% RSLogix 500 project PROJECT 4.RSS, saved by version 8.30.00.16 %
PROJECT "500"    % processor: Bul.1763 MicroLogix 1100 Series B %

PROGRAM FILES
  LAD 2 "MAIN"  4 rungs
  LAD 3 "IO"  7 rungs  % Digital Input %
  LAD 4 "CTRL"  13 rungs
  LAD 8 "CYCLE"  6 rungs

DATA FILES
  O0 OUTPUT  4 elements
  I1 INPUT  6 elements
  S2 STATUS  66 elements
  B3 BINARY  2 elements
  T4 TIMER  3 elements
  C5 COUNTER  1 elements
  R6 CONTROL  1 elements
  N7 INTEGER  1 elements
  F8 FLOAT  1 elements

LADDER 2 "MAIN"
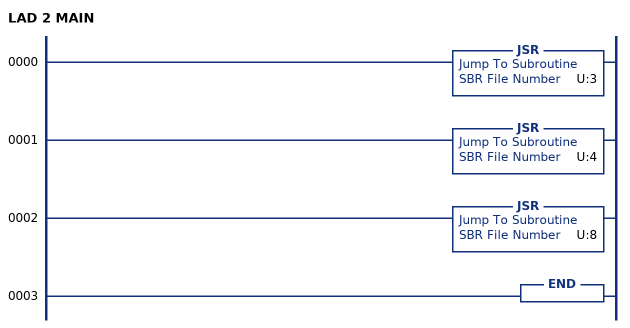
% Rung: 0 %
SOR JSR U:3 EOR
% Rung: 1 %
SOR JSR U:4 EOR
% Rung: 2 %
SOR JSR U:8 EOR
% Rung: 3 %
SOR END EOR

LADDER 3 "IO"    % Digital Input %
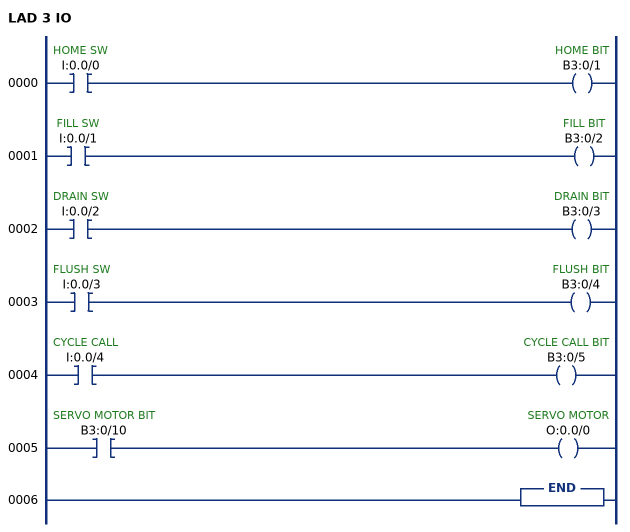
% Rung: 0 %
SOR XIC I:0.0/0 OTE B3:0/1 EOR
%   I:0.0/0  "HOME SW" %
%   B3:0/1  "HOME BIT" %
% Rung: 1 %
SOR XIC I:0.0/1 OTE B3:0/2 EOR
%   I:0.0/1  "FILL SW" %
%   B3:0/2  "FILL BIT" %
% Rung: 2 %
SOR XIC I:0.0/2 OTE B3:0/3 EOR
%   I:0.0/2  "DRAIN SW" %
%   B3:0/3  "DRAIN BIT" %
% Rung: 3 %
SOR XIC I:0.0/3 OTE B3:0/4 EOR
%   I:0.0/3  "FLUSH SW" %
%   B3:0/4  "FLUSH BIT" %
% Rung: 4 %
SOR XIC I:0.0/4 OTE B3:0/5 EOR
%   I:0.0/4  "CYCLE CALL" %
%   B3:0/5  "CYCLE CALL BIT" %
% Rung: 5 %
SOR XIC B3:0/10 OTE O:0.0/0 EOR
%   B3:0/10  "SERVO MOTOR BIT" %
%   O:0.0/0  "SERVO MOTOR" %
% Rung: 6 %
SOR END EOR

LADDER 4 "CTRL"
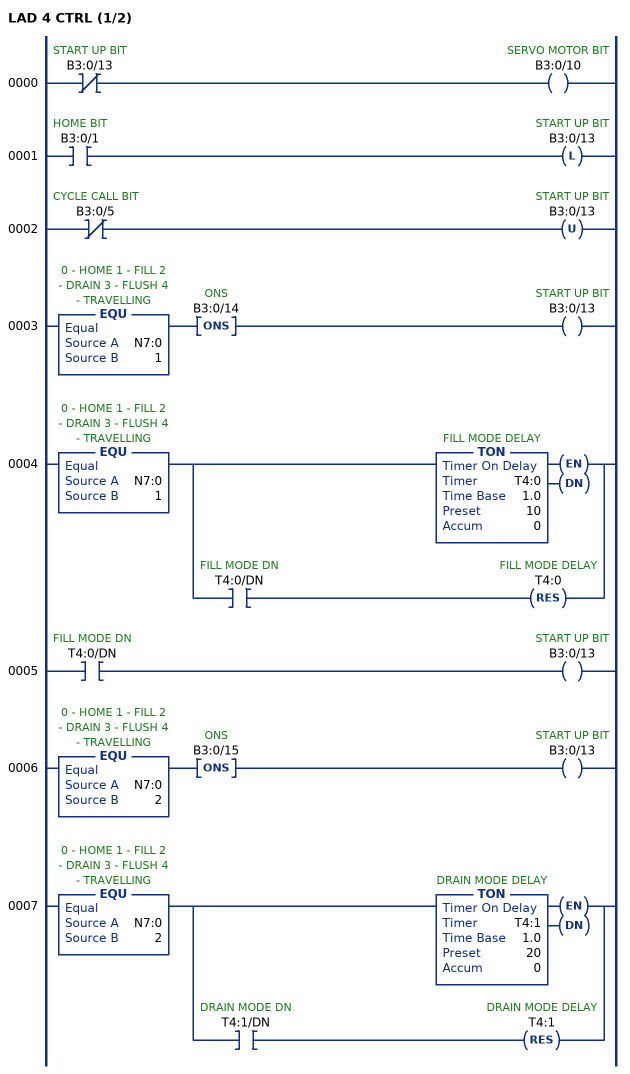
% Rung: 0 %
SOR XIO B3:0/13 OTE B3:0/10 EOR
%   B3:0/13  "START UP BIT" %
%   B3:0/10  "SERVO MOTOR BIT" %
% Rung: 1 %
SOR XIC B3:0/1 OTL B3:0/13 EOR
%   B3:0/1  "HOME BIT" %
%   B3:0/13  "START UP BIT" %
% Rung: 2 %
SOR XIO B3:0/5 OTU B3:0/13 EOR
%   B3:0/5  "CYCLE CALL BIT" %
%   B3:0/13  "START UP BIT" %
% Rung: 3 %
SOR EQU N7:0 1 ONS B3:0/14 OTE B3:0/13 EOR
%   N7:0  "0 - HOME 1 - FILL 2 - DRAIN 3 - FLUSH 4 - TRAVELLING" %
%   B3:0/14  "ONS" %
%   B3:0/13  "START UP BIT" %
% Rung: 4 %
SOR EQU N7:0 1 BST TON T4:0 1.0 10 0 NXB XIC T4:0/DN RES T4:0 BND EOR
%   N7:0  "0 - HOME 1 - FILL 2 - DRAIN 3 - FLUSH 4 - TRAVELLING" %
%   T4:0  "FILL MODE DELAY" %
%   T4:0/DN  "FILL MODE DN" %
% Rung: 5 %
SOR XIC T4:0/DN OTE B3:0/13 EOR
%   T4:0/DN  "FILL MODE DN" %
%   B3:0/13  "START UP BIT" %
% Rung: 6 %
SOR EQU N7:0 2 ONS B3:0/15 OTE B3:0/13 EOR
%   N7:0  "0 - HOME 1 - FILL 2 - DRAIN 3 - FLUSH 4 - TRAVELLING" %
%   B3:0/15  "ONS" %
%   B3:0/13  "START UP BIT" %
% Rung: 7 %
SOR EQU N7:0 2 BST TON T4:1 1.0 20 0 NXB XIC T4:1/DN RES T4:1 BND EOR
%   N7:0  "0 - HOME 1 - FILL 2 - DRAIN 3 - FLUSH 4 - TRAVELLING" %
%   T4:1  "DRAIN MODE DELAY" %
%   T4:1/DN  "DRAIN MODE DN" %

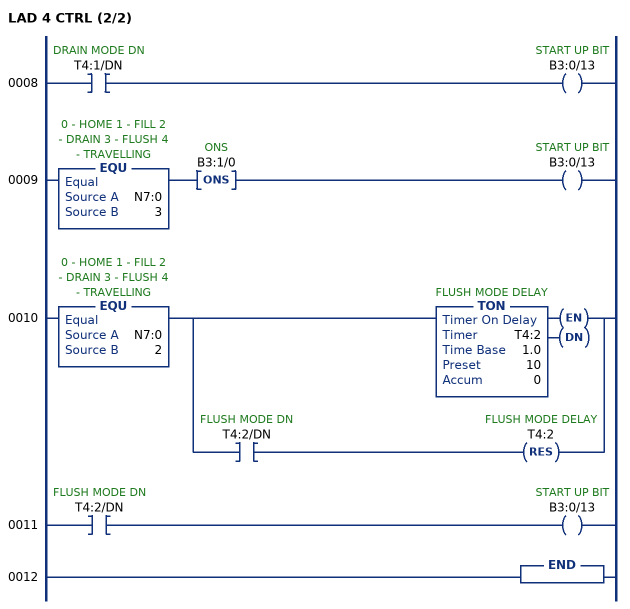
% Rung: 8 %
SOR XIC T4:1/DN OTE B3:0/13 EOR
%   T4:1/DN  "DRAIN MODE DN" %
%   B3:0/13  "START UP BIT" %
% Rung: 9 %
SOR EQU N7:0 3 ONS B3:1/0 OTE B3:0/13 EOR
%   N7:0  "0 - HOME 1 - FILL 2 - DRAIN 3 - FLUSH 4 - TRAVELLING" %
%   B3:1/0  "ONS" %
%   B3:0/13  "START UP BIT" %
% Rung: 10 %
SOR EQU N7:0 2 BST TON T4:2 1.0 10 0 NXB XIC T4:2/DN RES T4:2 BND EOR
%   N7:0  "0 - HOME 1 - FILL 2 - DRAIN 3 - FLUSH 4 - TRAVELLING" %
%   T4:2  "FLUSH MODE DELAY" %
%   T4:2/DN  "FLUSH MODE DN" %
% Rung: 11 %
SOR XIC T4:2/DN OTE B3:0/13 EOR
%   T4:2/DN  "FLUSH MODE DN" %
%   B3:0/13  "START UP BIT" %
% Rung: 12 %
SOR END EOR

LADDER 8 "CYCLE"
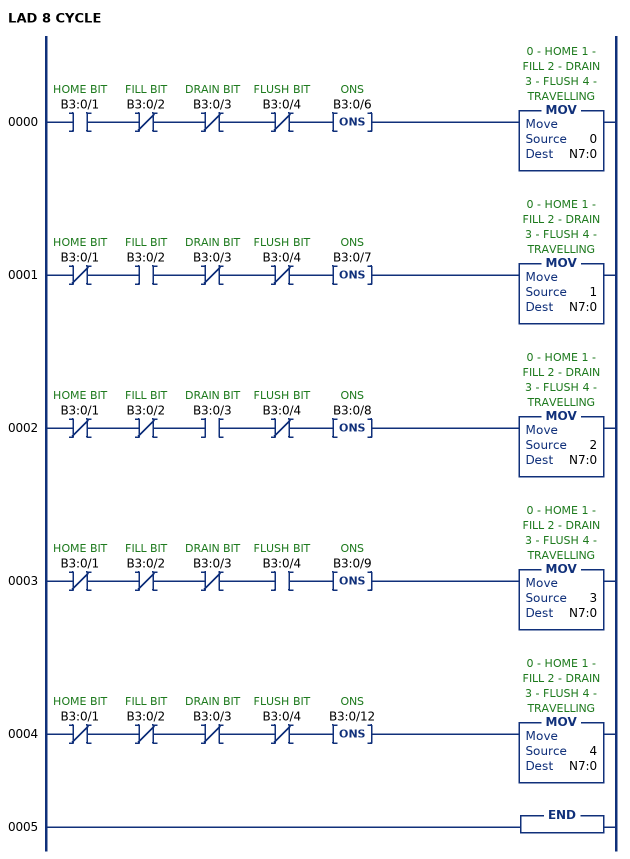
% Rung: 0 %
SOR XIC B3:0/1 XIO B3:0/2 XIO B3:0/3 XIO B3:0/4 ONS B3:0/6 MOV 0 N7:0 EOR
%   B3:0/1  "HOME BIT" %
%   B3:0/2  "FILL BIT" %
%   B3:0/3  "DRAIN BIT" %
%   B3:0/4  "FLUSH BIT" %
%   B3:0/6  "ONS" %
%   N7:0  "0 - HOME 1 - FILL 2 - DRAIN 3 - FLUSH 4 - TRAVELLING" %
% Rung: 1 %
SOR XIO B3:0/1 XIC B3:0/2 XIO B3:0/3 XIO B3:0/4 ONS B3:0/7 MOV 1 N7:0 EOR
%   B3:0/1  "HOME BIT" %
%   B3:0/2  "FILL BIT" %
%   B3:0/3  "DRAIN BIT" %
%   B3:0/4  "FLUSH BIT" %
%   B3:0/7  "ONS" %
%   N7:0  "0 - HOME 1 - FILL 2 - DRAIN 3 - FLUSH 4 - TRAVELLING" %
% Rung: 2 %
SOR XIO B3:0/1 XIO B3:0/2 XIC B3:0/3 XIO B3:0/4 ONS B3:0/8 MOV 2 N7:0 EOR
%   B3:0/1  "HOME BIT" %
%   B3:0/2  "FILL BIT" %
%   B3:0/3  "DRAIN BIT" %
%   B3:0/4  "FLUSH BIT" %
%   B3:0/8  "ONS" %
%   N7:0  "0 - HOME 1 - FILL 2 - DRAIN 3 - FLUSH 4 - TRAVELLING" %
% Rung: 3 %
SOR XIO B3:0/1 XIO B3:0/2 XIO B3:0/3 XIC B3:0/4 ONS B3:0/9 MOV 3 N7:0 EOR
%   B3:0/1  "HOME BIT" %
%   B3:0/2  "FILL BIT" %
%   B3:0/3  "DRAIN BIT" %
%   B3:0/4  "FLUSH BIT" %
%   B3:0/9  "ONS" %
%   N7:0  "0 - HOME 1 - FILL 2 - DRAIN 3 - FLUSH 4 - TRAVELLING" %
% Rung: 4 %
SOR XIO B3:0/1 XIO B3:0/2 XIO B3:0/3 XIO B3:0/4 ONS B3:0/12 MOV 4 N7:0 EOR
%   B3:0/1  "HOME BIT" %
%   B3:0/2  "FILL BIT" %
%   B3:0/3  "DRAIN BIT" %
%   B3:0/4  "FLUSH BIT" %
%   B3:0/12  "ONS" %
%   N7:0  "0 - HOME 1 - FILL 2 - DRAIN 3 - FLUSH 4 - TRAVELLING" %
% Rung: 5 %
SOR END EOR

OTHER DOCUMENTED ADDRESSES
  B3:0/11  "ONS"
  B3:1/1  "ONS"
  B3:1/2  "ONS"
  B3:2/1  "START UP BIT 1"
  I:0.0/5  "HH SWITCH"
  I:0.0/6  "H SWITCH"
  I:0.0/7  "LL SWITCH"
  I:0.0/8  "L SWITCH"
  I:1.0/1  "D_INPUT_1"
  I:3.0  "ANALOG INPUT 1"
  I:3.1  "ANALOG INPUT 2"
  I:3.2  "ANALOG INPUT 3"
  I:3.3  "ANALOG INPUT 4"
  I:3.4  "ANALOG INPUT 5"
  JSR  
  MOV  "DEVICE HOA 0 - OFF 1 - ON 2 - AUTO"
  O:0  "SERVO MOTOR"
  O:0.0/1  "DIGI DEVICE 1 OUTPUT"
  O:0.0/2  "DIGI DEVICE 2 OUTPUT"
  O:0.0/3  "DIGI DEVICE 3 OUTPUT"
  O:0.0/4  "DIGI DEVICE 4 OUTPUT"
  O:0.0/5  "DIGI DEVICE 5 OUTPUT"
  PFILE:4  "Digital Output"
  PFILE:5  "Analog Input"
  PFILE:6  "Analog Output"
  PFILE:8  "HAND_ON_AUTO MODE"
  SCP  "SCALE INPUT"

DATA TABLE (non-zero values as saved)
DATA T4
% .PRE .ACC %
% T4:0 % 10 0
% T4:1 % 20 0
% T4:2 % 10 0
